// TIA Portal V18 export
FUNCTION_BLOCK "AXIS_CMMT_V2_Motion_Control"   // FB22, LAD
TITLE = Description
{ S7_Optimized_Access := 'TRUE' }
VERSION : 0.1
// This is the motion function block used to control all the axes. Due to some differences in the control part for different types of motion and drives, there are additional conditions in some parts of the code.
// 
// Important things to check if the drive is not moving:
// - homing
// - motion lock from add ons (capping station, no go zones)
// - door sensors
// - operation mode
// - communication with the drives (Online access)
// stored: AutoNumber false, IsIECCheckEnabled false, IsRetainMemResEnabled false, MemoryReserve 100, SetENOAutomatically false, UDAEnableTagReadback false
   VAR_INPUT
      DriverType : String;   // CMMT; CMMS;
      EnableAxis : Bool;
      PrintingModeWebDB : Int;   // Used while executing the movement
      PositionWebDB : DInt;
      VelocityWebDB : Real;
      Stop : Bool;
      EmergencyStop : Bool;
      JogPos : Bool;
      JogNeg : Bool;
      AckError : Bool;
      ConfigEPos : DWord;
      PosMin : DInt;
      PosMax : DInt;
      Jogging : Bool;
      MarginSoft : DInt;
      MarginHard : DInt;
      MotionLock : Bool;   // Axis will not move is this bool is 0
      AXISEnabled : Bool;
      AXISPosOk : Bool;
      AXISReference : Bool;
      AXISAxisWarning : Bool;
      AXISAxisError : Bool;
      AXISLockout : Bool;
      AXISActVelocity : Real;
      AXISActPosition : DInt;
      AXISAxisAckSetpoint : Bool;
      AXISReady4Motion : Bool;
      AXISEposZSW1 : Word;
      AXISStatus : Word;
      JogStartPos : DInt;   // Limit for jogging
      JogEndPos : DInt;   // Limit for jogging
      AxisType : Int;   // Axis Type: 1 - X; 2 - Y; 3 - Z1; 4 - Z2
      YPosition : DInt;
      PositionDelay : Bool;   // Delay to make it easier to confirm that the motion was finished
      NoGoZoneActive : Bool;   // 1 to activate no go zone
      NoGoZoneHomingPermission : Bool;
      NoGoZoneMovePermission : Bool;
      NoGoZoneJogPosPermission : Bool;
      NoGoZoneJogNegPermission : Bool;
      RMPositioningError : DInt := 5;   // Input Relativer Motion Position Error that we accept
      MachineStart : Bool;
   END_VAR
   VAR_OUTPUT
      Status : Word;
      Overrange : Bool;
      Ready : Bool;
      DriveMoving : Bool;
      DriveStop : Bool;
      Standstill : Bool;
      MC : Bool;
      AXISModePos : Int;
      AXISEnableAxis : Bool;
      AXISCancelTraversing : Bool;
      AXISIntermediateStop : Bool;
      AXISJog1 : Bool;
      AXISJog2 : Bool;
      AXISAckError : Bool;
      AXISExecuteMode : Bool;
      AXISPosition : DInt;
      AXISVelocity : Real;
      AXISConfigEpos : DWord;
      AXISRelative : Bool;
      AXISHoming : Bool;
      FinishTask_Delay : Bool;
   END_VAR
   VAR_IN_OUT
      StartTask : Bool;
      Execute : Bool;
      Homing : Bool;
      Printing : Bool;
   END_VAR
   VAR
      ExecutingMemory : Bool;
      HomingMemory : Bool;
      TaskMemory : Bool;
      ModePos : Int := 4;
      PosOk : Bool;
      Reference : Bool;
      PositionInternal : DInt;
      LockoutInternal : Bool;
      RelativeMode : Bool;   // Mode 1
      AbsoluteMode : Bool;   // Mode 2
      TaskFinished : Bool;
      JoggingXPermission : Bool;
      JoggingYPermission : Bool;
      JoggingPOSZ1Z2Permission : Bool;
      JoggingNEGZ1Z2Permission : Bool;
      JoggingPosMax : DInt;
      JoggingPosMin : DInt;
      JoggingPositionCorrection : DInt := 1500;
      ProfinetDisconnected : Bool;
      PositionStepPlus : DInt;
      CMMT : Bool;
      CMMS : Bool;
      RMStepStartPosition : DInt;   // Relative Motion Step Start Position
      RMPredictedPosition : DInt;   // Relative Motion Predicted Position
      RMFinalPosition : DInt;   // Relative Motion Final Position
      RMLastStepPositionError : DInt;   // Relative Motion Last Step Position Error
      RMStartTaskM01 : Bool;   // Relative Motion Start Task M Positive
      RMStartTaksM02 : Bool;   // Relative Motion Start Task M Negative
      RMStepRangePlus : DInt;
      RMStepRangeMinus : DInt;
      RelativeDirectionInRange : Bool;
   END_VAR
   VAR_TEMP
      RelativeModeHomingM : Bool;
      Jog1_pos : Bool;   // Jog positive direction
      Jog2_neg : Bool;   // Jog negative direction
      Memory1 : Bool;
      Memory2 : Bool;
      PosMinSoft : DInt;
      PosMaxSoft : DInt;
      InternalError : Bool;
      InternalWarning : Bool;
      ExecuteBusy : Bool;
      ExecutingInternal : Bool;
      HomingInternal : Bool;
      TaskInternal : Bool;
      Position_Plus : DInt;
      Position_Minus : DInt;
      TestFinished : Bool;
   END_VAR
   VAR CONSTANT
      Position_Error : DInt := 10;
   END_VAR
   VAR_TEMP   // added for the SCL form of the ladder/FBD networks
      _w1 : Bool;
      _w2 : Bool;
      _w3 : Bool;
   END_VAR
BEGIN

REGION Network 1: Checking driver type
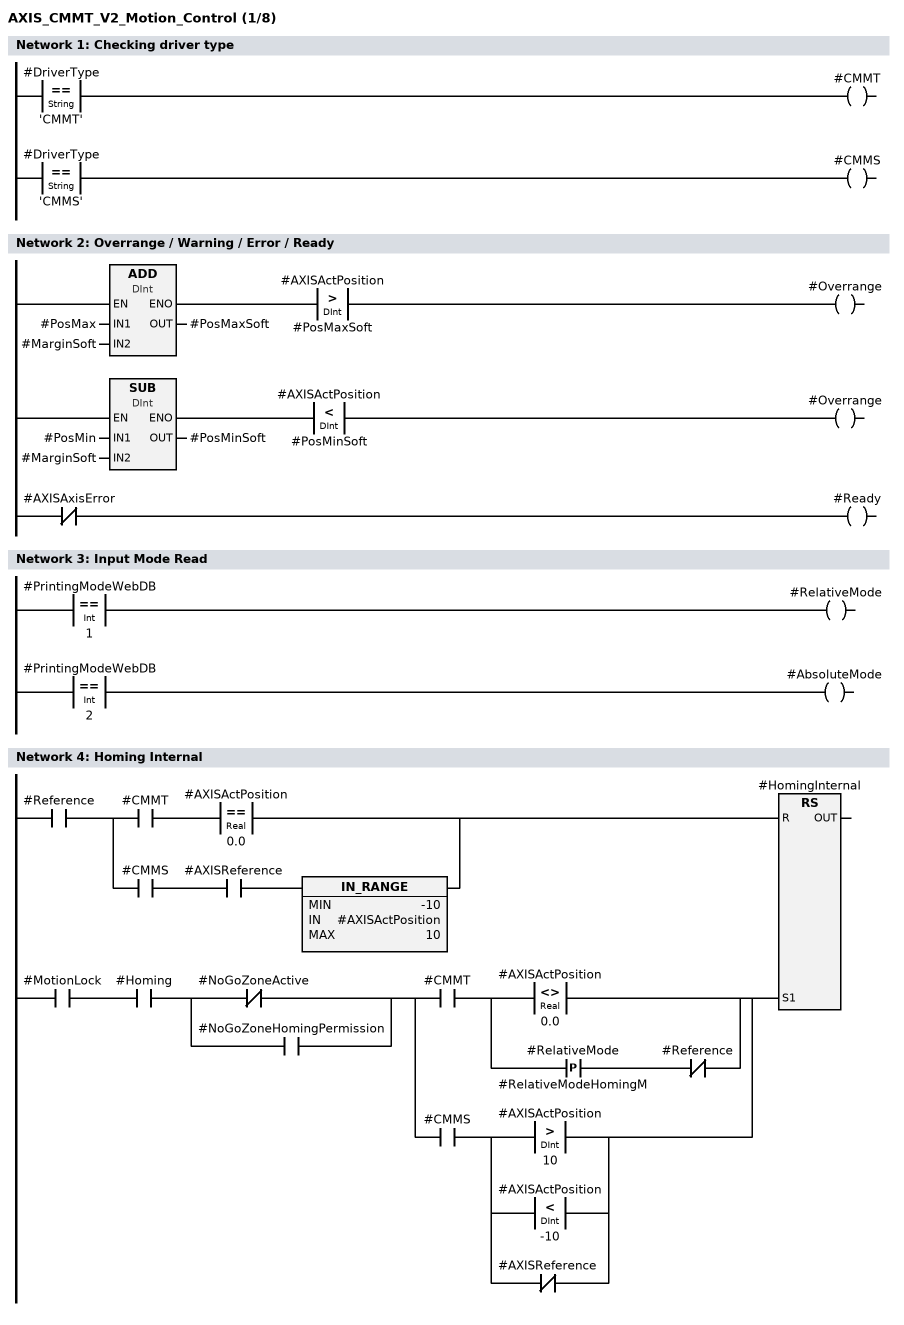
   RUNG wire#powerrail
      { S7_Templates := "SrcType := String" } EQ_Contact(in1 := #DriverType, in2 := 'CMMT')
      Coil( #CMMT )
   END_RUNG
   RUNG wire#powerrail
      { S7_Templates := "SrcType := String" } EQ_Contact(in1 := #DriverType, in2 := 'CMMS')
      Coil( #CMMS )
   END_RUNG
   // the same network as SCL:
   #CMMT := #DriverType = 'CMMT';
   #CMMS := #DriverType = 'CMMS';
END_REGION

REGION Network 2: Overrange / Warning / Error / Ready
   RUNG wire#powerrail
      { S7_Templates := "SrcType := DInt" } Add(in1 := #PosMax, in2 := #MarginSoft, out => #PosMaxSoft)
      { S7_Templates := "SrcType := DInt" } GT_Contact(in1 := #AXISActPosition, in2 := #PosMaxSoft)
      Coil( #Overrange )
   END_RUNG
   RUNG wire#powerrail
      { S7_Templates := "SrcType := DInt" } Sub(in1 := #PosMin, in2 := #MarginSoft, out => #PosMinSoft)
      { S7_Templates := "SrcType := DInt" } LT_Contact(in1 := #AXISActPosition, in2 := #PosMinSoft)
      Coil( #Overrange )
   END_RUNG
   RUNG wire#powerrail
      I_Contact( #AXISAxisError )
      Coil( #Ready )
   END_RUNG
   // the same network as SCL:
   #PosMaxSoft := #PosMax + #MarginSoft;
   #Overrange := #AXISActPosition > #PosMaxSoft;
   #PosMinSoft := #PosMin - #MarginSoft;
   #Overrange := #AXISActPosition < #PosMinSoft;
   #Ready := NOT #AXISAxisError;
END_REGION

REGION Network 3: Input Mode Read
   RUNG wire#powerrail
      { S7_Templates := "SrcType := Int" } EQ_Contact(in1 := #PrintingModeWebDB, in2 := 1)
      Coil( #RelativeMode )
   END_RUNG
   RUNG wire#powerrail
      { S7_Templates := "SrcType := Int" } EQ_Contact(in1 := #PrintingModeWebDB, in2 := 2)
      Coil( #AbsoluteMode )
   END_RUNG
   // the same network as SCL:
   #RelativeMode := #PrintingModeWebDB = 1;
   #AbsoluteMode := #PrintingModeWebDB = 2;
END_REGION

REGION Network 4: Homing Internal
   RUNG wire#powerrail
      Contact( #Reference )
      wire#w1
      Contact( #CMMT )
      { S7_Templates := "SrcType := Real" } EQ_Contact(in1 := #AXISActPosition, in2 := 0.0)
      wire#w2
      S_RS(operand := #HomingInternal, s1 := wire#w7)
   END_RUNG
   RUNG wire#w1
      Contact( #CMMS )
      Contact( #AXISReference )
      { S7_Templates := "SrcType := DInt" } InRange(min := -10, in := #AXISActPosition, max := 10)
   END_RUNG wire#w2
   RUNG wire#powerrail
      Contact( #MotionLock )
      Contact( #Homing )
      wire#w3
      I_Contact( #NoGoZoneActive )
      wire#w4
      Contact( #CMMT )
      wire#w5
      { S7_Templates := "SrcType := Real" } NE_Contact(in1 := #AXISActPosition, in2 := 0.0)
   END_RUNG wire#w7
   RUNG wire#w3
      Contact( #NoGoZoneHomingPermission )
   END_RUNG wire#w4
   RUNG wire#w5
      P_Contact(operand := #RelativeMode, bit := #RelativeModeHomingM)
      I_Contact( #Reference )
   END_RUNG wire#w7
   RUNG wire#w4
      Contact( #CMMS )
      wire#w6
      { S7_Templates := "SrcType := DInt" } GT_Contact(in1 := #AXISActPosition, in2 := 10)
   END_RUNG wire#w7
   RUNG wire#w6
      { S7_Templates := "SrcType := DInt" } LT_Contact(in1 := #AXISActPosition, in2 := -10)
   END_RUNG wire#w7
   RUNG wire#w6
      I_Contact( #AXISReference )
   END_RUNG wire#w7
   // the same network as SCL:
   #_w1 := #MotionLock AND #Homing AND (NOT #NoGoZoneActive OR #NoGoZoneHomingPermission) AND #CMMT AND #RelativeMode AND NOT #RelativeModeHomingM;   // rising edge of #RelativeMode
   #RelativeModeHomingM := #RelativeMode;
   IF #Reference AND ((#CMMT AND (#AXISActPosition = 0.0)) OR (#CMMS AND #AXISReference AND (-10 <= #AXISActPosition) AND (#AXISActPosition <= 10))) THEN
       #HomingInternal := FALSE;   // RS flip-flop
   END_IF;
   IF (#MotionLock AND #Homing AND (NOT #NoGoZoneActive OR #NoGoZoneHomingPermission) AND #CMMT AND (#AXISActPosition <> 0.0)) OR (#_w1 AND NOT #Reference) OR (#MotionLock AND #Homing AND (NOT #NoGoZoneActive OR #NoGoZoneHomingPermission) AND #CMMS AND ((#AXISActPosition > 10) OR (#AXISActPosition < (-10)) OR NOT #AXISReference)) THEN
       #HomingInternal := TRUE;
   END_IF;
END_REGION

REGION Network 5: Status Behavior
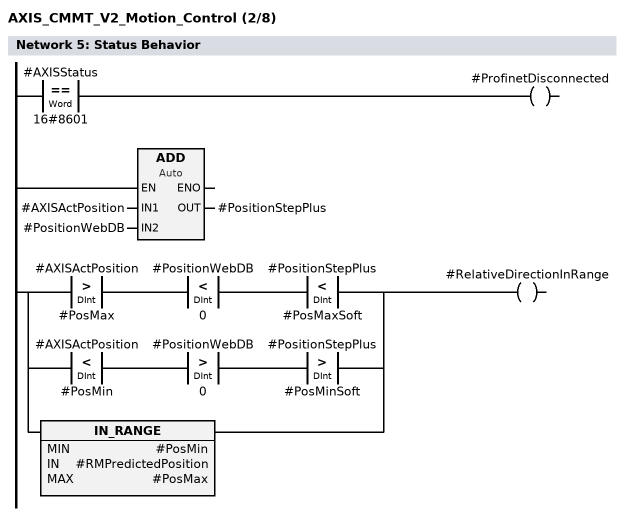
   RUNG wire#powerrail
      { S7_Templates := "SrcType := Word" } EQ_Contact(in1 := #AXISStatus, in2 := 16#8601)
      Coil( #ProfinetDisconnected )
   END_RUNG
   RUNG wire#powerrail
      Add(in1 := #AXISActPosition, in2 := #PositionWebDB, out => #PositionStepPlus)
   END_RUNG
   RUNG wire#powerrail
      { S7_Templates := "SrcType := DInt" } GT_Contact(in1 := #AXISActPosition, in2 := #PosMax)
      { S7_Templates := "SrcType := DInt" } LT_Contact(in1 := #PositionWebDB, in2 := 0)
      { S7_Templates := "SrcType := DInt" } LT_Contact(in1 := #PositionStepPlus, in2 := #PosMaxSoft)
      wire#w1
      Coil( #RelativeDirectionInRange )
   END_RUNG
   RUNG wire#powerrail
      { S7_Templates := "SrcType := DInt" } LT_Contact(in1 := #AXISActPosition, in2 := #PosMin)
      { S7_Templates := "SrcType := DInt" } GT_Contact(in1 := #PositionWebDB, in2 := 0)
      { S7_Templates := "SrcType := DInt" } GT_Contact(in1 := #PositionStepPlus, in2 := #PosMinSoft)
   END_RUNG wire#w1
   RUNG wire#powerrail
      { S7_Templates := "SrcType := DInt" } InRange(min := #PosMin, in := #RMPredictedPosition, max := #PosMax)
   END_RUNG wire#w1
   // the same network as SCL:
   #ProfinetDisconnected := #AXISStatus = 16#8601;
   #PositionStepPlus := #AXISActPosition + #PositionWebDB;
   #RelativeDirectionInRange := ((#AXISActPosition > #PosMax) AND (#PositionWebDB < 0) AND (#PositionStepPlus < #PosMaxSoft)) OR ((#AXISActPosition < #PosMin) AND (#PositionWebDB > 0) AND (#PositionStepPlus > #PosMinSoft)) OR ((#PosMin <= #RMPredictedPosition) AND (#RMPredictedPosition <= #PosMax));
END_REGION

REGION Network 6: Task Internal
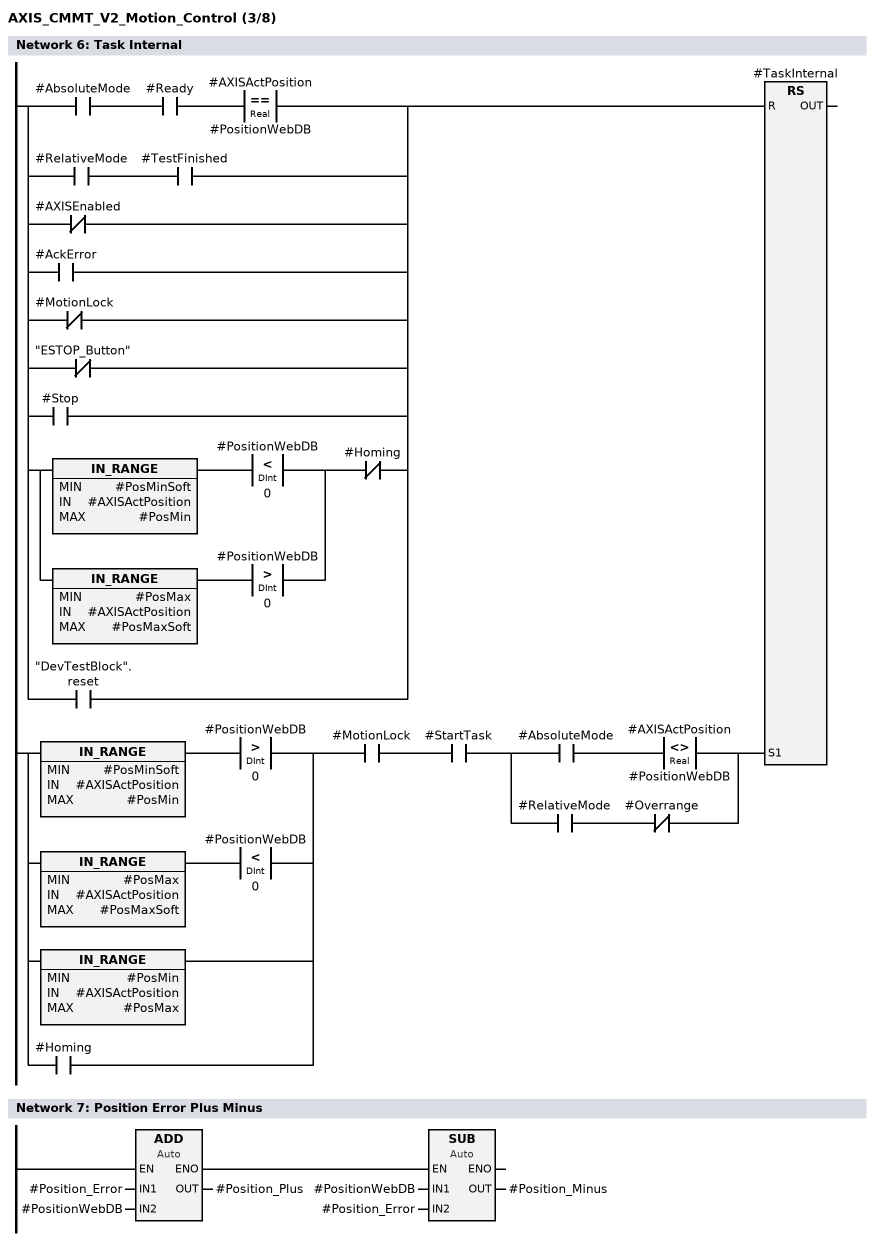
   RUNG wire#powerrail
      Contact( #AbsoluteMode )
      Contact( #Ready )
      { S7_Templates := "SrcType := Real" } EQ_Contact(in1 := #AXISActPosition, in2 := #PositionWebDB)
      wire#w1
      S_RS(operand := #TaskInternal, s1 := wire#w5)
   END_RUNG
   RUNG wire#powerrail
      Contact( #RelativeMode )
      Contact( #TestFinished )
   END_RUNG wire#w1
   RUNG wire#powerrail
      I_Contact( #AXISEnabled )
   END_RUNG wire#w1
   RUNG wire#powerrail
      Contact( #AckError )
   END_RUNG wire#w1
   RUNG wire#powerrail
      I_Contact( #MotionLock )
   END_RUNG wire#w1
   RUNG wire#powerrail
      I_Contact( "ESTOP_Button" )
   END_RUNG wire#w1
   RUNG wire#powerrail
      Contact( #Stop )
   END_RUNG wire#w1
   RUNG wire#powerrail
      { S7_Templates := "SrcType := DInt" } InRange(min := #PosMinSoft, in := #AXISActPosition, max := #PosMin)
      { S7_Templates := "SrcType := DInt" } LT_Contact(in1 := #PositionWebDB, in2 := 0)
      wire#w2
      I_Contact( #Homing )
   END_RUNG wire#w1
   RUNG wire#powerrail
      { S7_Templates := "SrcType := DInt" } InRange(min := #PosMax, in := #AXISActPosition, max := #PosMaxSoft)
      { S7_Templates := "SrcType := DInt" } GT_Contact(in1 := #PositionWebDB, in2 := 0)
   END_RUNG wire#w2
   RUNG wire#powerrail
      Contact( "DevTestBlock".reset )
   END_RUNG wire#w1
   RUNG wire#powerrail
      { S7_Templates := "SrcType := DInt" } InRange(min := #PosMinSoft, in := #AXISActPosition, max := #PosMin)
      { S7_Templates := "SrcType := DInt" } GT_Contact(in1 := #PositionWebDB, in2 := 0)
      wire#w3
      Contact( #MotionLock )
      Contact( #StartTask )
      wire#w4
      Contact( #AbsoluteMode )
      { S7_Templates := "SrcType := Real" } NE_Contact(in1 := #AXISActPosition, in2 := #PositionWebDB)
   END_RUNG wire#w5
   RUNG wire#powerrail
      { S7_Templates := "SrcType := DInt" } InRange(min := #PosMax, in := #AXISActPosition, max := #PosMaxSoft)
      { S7_Templates := "SrcType := DInt" } LT_Contact(in1 := #PositionWebDB, in2 := 0)
   END_RUNG wire#w3
   RUNG wire#powerrail
      { S7_Templates := "SrcType := DInt" } InRange(min := #PosMin, in := #AXISActPosition, max := #PosMax)
   END_RUNG wire#w3
   RUNG wire#powerrail
      Contact( #Homing )
   END_RUNG wire#w3
   RUNG wire#w4
      Contact( #RelativeMode )
      I_Contact( #Overrange )
   END_RUNG wire#w5
   // the same network as SCL:
   IF (#AbsoluteMode AND #Ready AND (#AXISActPosition = #PositionWebDB)) OR (#RelativeMode AND #TestFinished) OR NOT #AXISEnabled OR #AckError OR NOT #MotionLock OR NOT "ESTOP_Button" OR #Stop OR ((((#PosMinSoft <= #AXISActPosition) AND (#AXISActPosition <= #PosMin) AND (#PositionWebDB < 0)) OR ((#PosMax <= #AXISActPosition) AND (#AXISActPosition <= #PosMaxSoft) AND (#PositionWebDB > 0))) AND NOT #Homing) OR "DevTestBlock".reset THEN
       #TaskInternal := FALSE;   // RS flip-flop
   END_IF;
   IF (((#PosMinSoft <= #AXISActPosition) AND (#AXISActPosition <= #PosMin) AND (#PositionWebDB > 0)) OR ((#PosMax <= #AXISActPosition) AND (#AXISActPosition <= #PosMaxSoft) AND (#PositionWebDB < 0)) OR ((#PosMin <= #AXISActPosition) AND (#AXISActPosition <= #PosMax)) OR #Homing) AND #MotionLock AND #StartTask AND ((#AbsoluteMode AND (#AXISActPosition <> #PositionWebDB)) OR (#RelativeMode AND NOT #Overrange)) THEN
       #TaskInternal := TRUE;
   END_IF;
END_REGION

REGION Network 7: Position Error Plus Minus
   RUNG wire#powerrail
      Add(in1 := #Position_Error, in2 := #PositionWebDB, out => #Position_Plus)
      Sub(in1 := #PositionWebDB, in2 := #Position_Error, out => #Position_Minus)
   END_RUNG
   // the same network as SCL:
   #Position_Plus := #Position_Error + #PositionWebDB;
   #Position_Minus := #PositionWebDB - #Position_Error;
END_REGION

REGION Network 8: Execute Internal
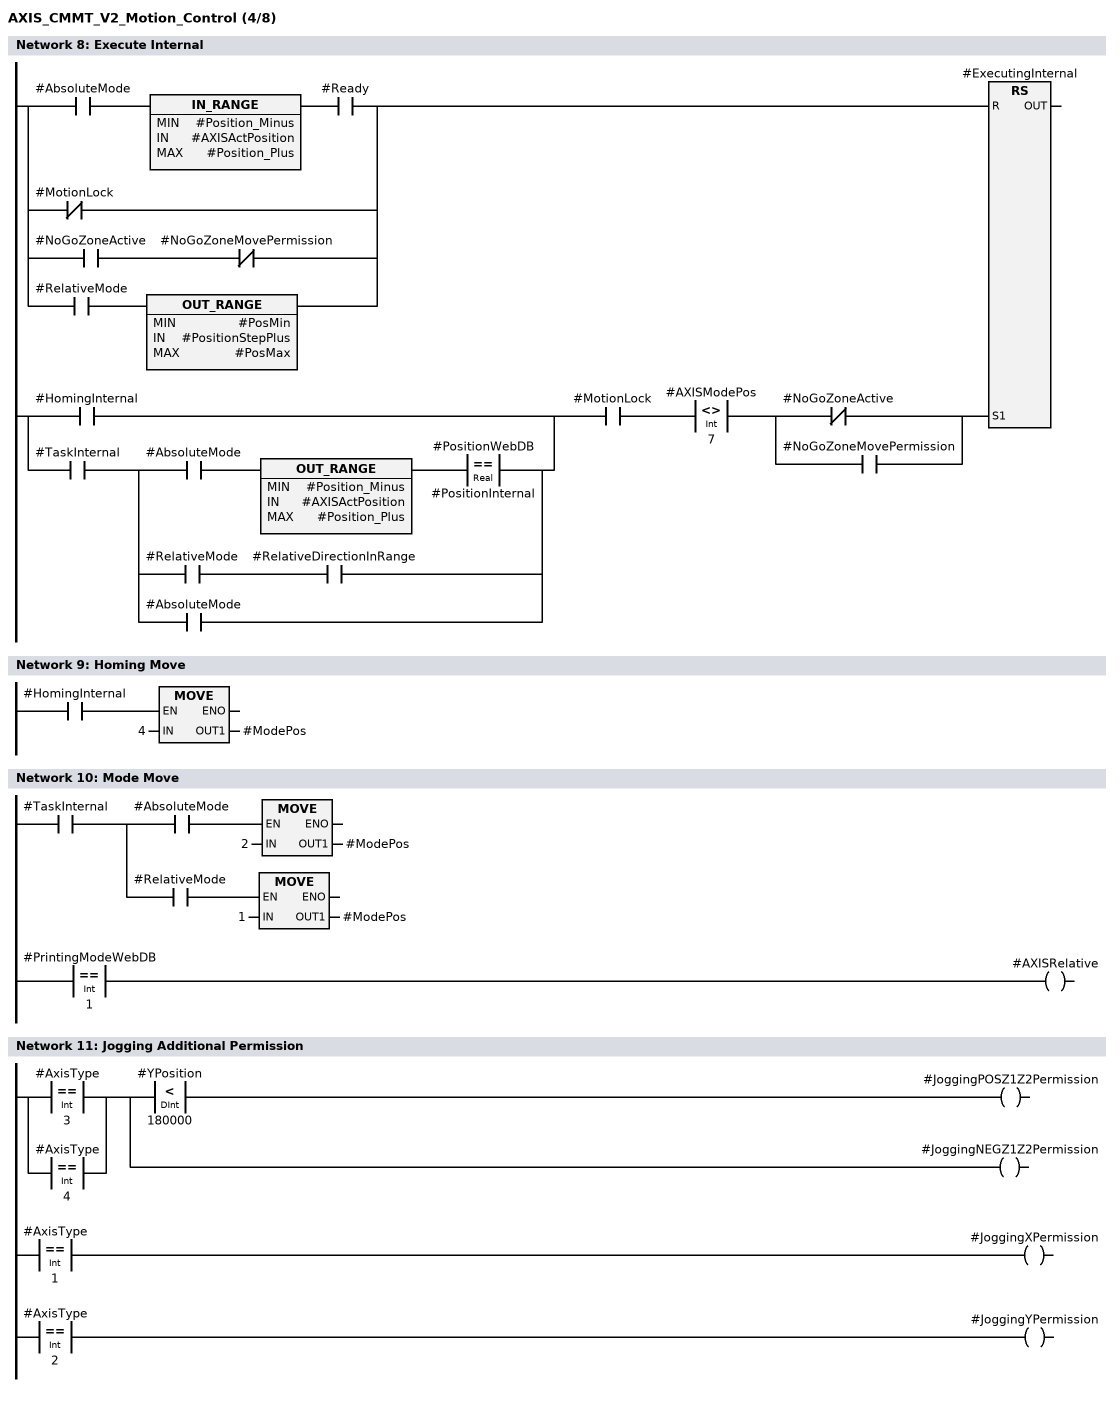
   IF (#AbsoluteMode AND (#Position_Minus <= #AXISActPosition) AND (#AXISActPosition <= #Position_Plus) AND #Ready) OR NOT #MotionLock OR (#NoGoZoneActive AND NOT #NoGoZoneMovePermission) OR (#RelativeMode AND ((#PositionStepPlus < #PosMin) OR (#PositionStepPlus > #PosMax))) THEN
       #ExecutingInternal := FALSE;   // RS flip-flop
   END_IF;
   IF (#HomingInternal OR (#TaskInternal AND ((#AbsoluteMode AND ((#AXISActPosition < #Position_Minus) OR (#AXISActPosition > #Position_Plus)) AND (#PositionWebDB = #PositionInternal)) OR (#RelativeMode AND #RelativeDirectionInRange) OR #AbsoluteMode))) AND #MotionLock AND (#AXISModePos <> 7) AND (NOT #NoGoZoneActive OR #NoGoZoneMovePermission) THEN
       #ExecutingInternal := TRUE;
   END_IF;
END_REGION

REGION Network 9: Homing Move
   RUNG wire#powerrail
      Contact( #HomingInternal )
      Move(in := 4, out1 => #ModePos)
   END_RUNG
   // the same network as SCL:
   IF #HomingInternal THEN #ModePos := 4; END_IF;
END_REGION

REGION Network 10: Mode Move
   RUNG wire#powerrail
      Contact( #TaskInternal )
      wire#w1
      Contact( #AbsoluteMode )
      Move(in := 2, out1 => #ModePos)
   END_RUNG
   RUNG wire#w1
      Contact( #RelativeMode )
      Move(in := 1, out1 => #ModePos)
   END_RUNG
   RUNG wire#powerrail
      { S7_Templates := "SrcType := Int" } EQ_Contact(in1 := #PrintingModeWebDB, in2 := 1)
      Coil( #AXISRelative )
   END_RUNG
   // the same network as SCL:
   IF #TaskInternal AND #AbsoluteMode THEN #ModePos := 2; END_IF;
   IF #TaskInternal AND #RelativeMode THEN #ModePos := 1; END_IF;
   #AXISRelative := #PrintingModeWebDB = 1;
END_REGION

REGION Network 11: Jogging Additional Permission
   RUNG wire#powerrail
      { S7_Templates := "SrcType := Int" } EQ_Contact(in1 := #AxisType, in2 := 3)
      wire#w1
      { S7_Templates := "SrcType := DInt" } LT_Contact(in1 := #YPosition, in2 := 180000)
      Coil( #JoggingPOSZ1Z2Permission )
   END_RUNG
   RUNG wire#powerrail
      { S7_Templates := "SrcType := Int" } EQ_Contact(in1 := #AxisType, in2 := 4)
   END_RUNG wire#w1
   RUNG wire#w1
      Coil( #JoggingNEGZ1Z2Permission )
   END_RUNG
   RUNG wire#powerrail
      { S7_Templates := "SrcType := Int" } EQ_Contact(in1 := #AxisType, in2 := 1)
      Coil( #JoggingXPermission )
   END_RUNG
   RUNG wire#powerrail
      { S7_Templates := "SrcType := Int" } EQ_Contact(in1 := #AxisType, in2 := 2)
      Coil( #JoggingYPermission )
   END_RUNG
   // the same network as SCL:
   #_w1 := (#AxisType = 3) OR (#AxisType = 4);
   #JoggingPOSZ1Z2Permission := #_w1 AND (#YPosition < 180000);
   #JoggingNEGZ1Z2Permission := #_w1;
   #JoggingXPermission := #AxisType = 1;
   #JoggingYPermission := #AxisType = 2;
END_REGION

REGION Network 12: Jogging Limit Change
   // Changed jogging limits to prevent overshooting
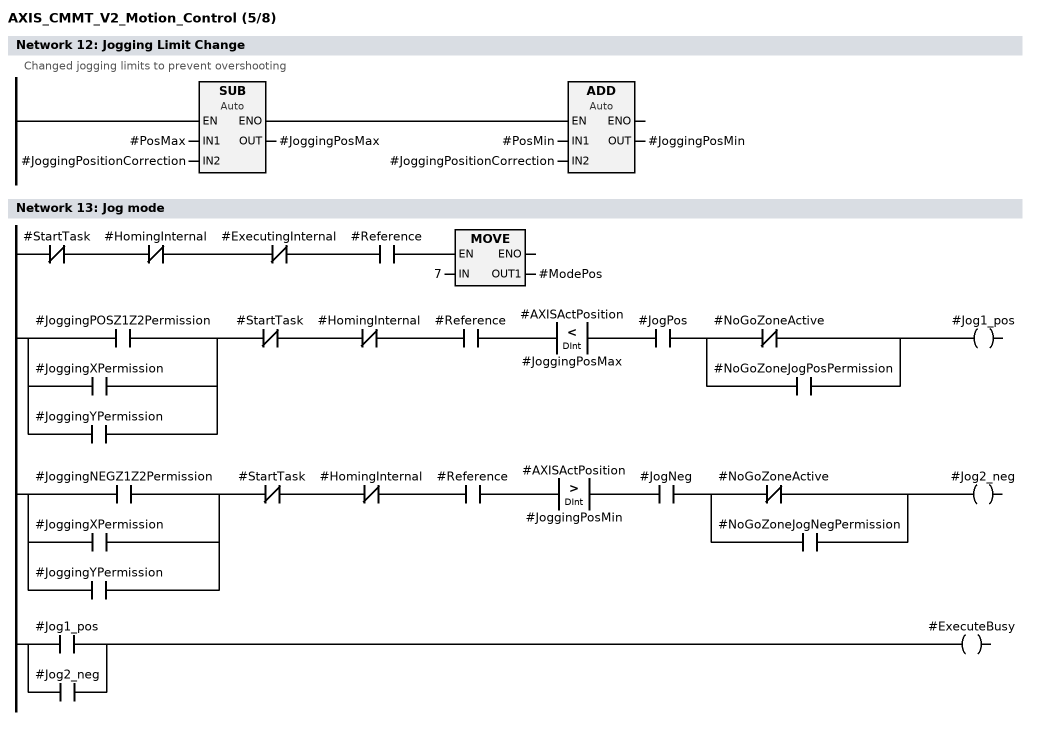
   RUNG wire#powerrail
      Sub(in1 := #PosMax, in2 := #JoggingPositionCorrection, out => #JoggingPosMax)
      Add(in1 := #PosMin, in2 := #JoggingPositionCorrection, out => #JoggingPosMin)
   END_RUNG
   // the same network as SCL:
   #JoggingPosMax := #PosMax - #JoggingPositionCorrection;
   #JoggingPosMin := #PosMin + #JoggingPositionCorrection;
END_REGION

REGION Network 13: Jog mode
   RUNG wire#powerrail
      I_Contact( #StartTask )
      I_Contact( #HomingInternal )
      I_Contact( #ExecutingInternal )
      Contact( #Reference )
      Move(in := 7, out1 => #ModePos)
   END_RUNG
   RUNG wire#powerrail
      Contact( #JoggingPOSZ1Z2Permission )
      wire#w1
      I_Contact( #StartTask )
      I_Contact( #HomingInternal )
      Contact( #Reference )
      { S7_Templates := "SrcType := DInt" } LT_Contact(in1 := #AXISActPosition, in2 := #JoggingPosMax)
      Contact( #JogPos )
      wire#w2
      I_Contact( #NoGoZoneActive )
      wire#w3
      Coil( #Jog1_pos )
   END_RUNG
   RUNG wire#powerrail
      Contact( #JoggingXPermission )
   END_RUNG wire#w1
   RUNG wire#powerrail
      Contact( #JoggingYPermission )
   END_RUNG wire#w1
   RUNG wire#w2
      Contact( #NoGoZoneJogPosPermission )
   END_RUNG wire#w3
   RUNG wire#powerrail
      Contact( #JoggingNEGZ1Z2Permission )
      wire#w4
      I_Contact( #StartTask )
      I_Contact( #HomingInternal )
      Contact( #Reference )
      { S7_Templates := "SrcType := DInt" } GT_Contact(in1 := #AXISActPosition, in2 := #JoggingPosMin)
      Contact( #JogNeg )
      wire#w5
      I_Contact( #NoGoZoneActive )
      wire#w6
      Coil( #Jog2_neg )
   END_RUNG
   RUNG wire#powerrail
      Contact( #JoggingXPermission )
   END_RUNG wire#w4
   RUNG wire#powerrail
      Contact( #JoggingYPermission )
   END_RUNG wire#w4
   RUNG wire#w5
      Contact( #NoGoZoneJogNegPermission )
   END_RUNG wire#w6
   RUNG wire#powerrail
      Contact( #Jog1_pos )
      wire#w7
      Coil( #ExecuteBusy )
   END_RUNG
   RUNG wire#powerrail
      Contact( #Jog2_neg )
   END_RUNG wire#w7
   // the same network as SCL:
   IF NOT #StartTask AND NOT #HomingInternal AND NOT #ExecutingInternal AND #Reference THEN
       #ModePos := 7;
   END_IF;
   #Jog1_pos := (#JoggingPOSZ1Z2Permission OR #JoggingXPermission OR #JoggingYPermission) AND NOT #StartTask AND NOT #HomingInternal AND #Reference AND (#AXISActPosition < #JoggingPosMax) AND #JogPos AND (NOT #NoGoZoneActive OR #NoGoZoneJogPosPermission);
   #Jog2_neg := (#JoggingNEGZ1Z2Permission OR #JoggingXPermission OR #JoggingYPermission) AND NOT #StartTask AND NOT #HomingInternal AND #Reference AND (#AXISActPosition > #JoggingPosMin) AND #JogNeg AND (NOT #NoGoZoneActive OR #NoGoZoneJogNegPermission);
   #ExecuteBusy := #Jog1_pos OR #Jog2_neg;
END_REGION

REGION Network 14: Motion Block Control
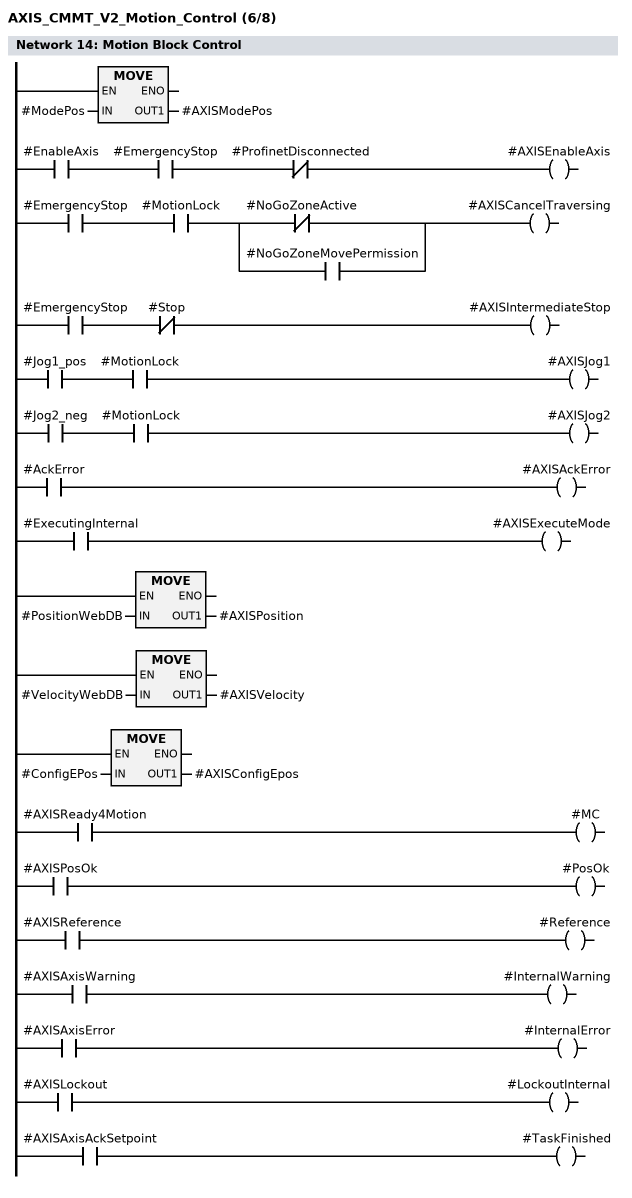
   RUNG wire#powerrail
      Move(in := #ModePos, out1 => #AXISModePos)
   END_RUNG
   RUNG wire#powerrail
      Contact( #EnableAxis )
      Contact( #EmergencyStop )
      I_Contact( #ProfinetDisconnected )
      Coil( #AXISEnableAxis )
   END_RUNG
   RUNG wire#powerrail
      Contact( #EmergencyStop )
      Contact( #MotionLock )
      wire#w1
      I_Contact( #NoGoZoneActive )
      wire#w2
      Coil( #AXISCancelTraversing )
   END_RUNG
   RUNG wire#w1
      Contact( #NoGoZoneMovePermission )
   END_RUNG wire#w2
   RUNG wire#powerrail
      Contact( #EmergencyStop )
      I_Contact( #Stop )
      Coil( #AXISIntermediateStop )
   END_RUNG
   RUNG wire#powerrail
      Contact( #Jog1_pos )
      Contact( #MotionLock )
      Coil( #AXISJog1 )
   END_RUNG
   RUNG wire#powerrail
      Contact( #Jog2_neg )
      Contact( #MotionLock )
      Coil( #AXISJog2 )
   END_RUNG
   RUNG wire#powerrail
      Contact( #AckError )
      Coil( #AXISAckError )
   END_RUNG
   RUNG wire#powerrail
      Contact( #ExecutingInternal )
      Coil( #AXISExecuteMode )
   END_RUNG
   RUNG wire#powerrail
      Move(in := #PositionWebDB, out1 => #AXISPosition)
   END_RUNG
   RUNG wire#powerrail
      Move(in := #VelocityWebDB, out1 => #AXISVelocity)
   END_RUNG
   RUNG wire#powerrail
      Move(in := #ConfigEPos, out1 => #AXISConfigEpos)
   END_RUNG
   RUNG wire#powerrail
      Contact( #AXISReady4Motion )
      Coil( #MC )
   END_RUNG
   RUNG wire#powerrail
      Contact( #AXISPosOk )
      Coil( #PosOk )
   END_RUNG
   RUNG wire#powerrail
      Contact( #AXISReference )
      Coil( #Reference )
   END_RUNG
   RUNG wire#powerrail
      Contact( #AXISAxisWarning )
      Coil( #InternalWarning )
   END_RUNG
   RUNG wire#powerrail
      Contact( #AXISAxisError )
      Coil( #InternalError )
   END_RUNG
   RUNG wire#powerrail
      Contact( #AXISLockout )
      Coil( #LockoutInternal )
   END_RUNG
   RUNG wire#powerrail
      Contact( #AXISAxisAckSetpoint )
      Coil( #TaskFinished )
   END_RUNG
   // the same network as SCL:
   #AXISModePos := #ModePos;
   #AXISEnableAxis := #EnableAxis AND #EmergencyStop AND NOT #ProfinetDisconnected;
   #AXISCancelTraversing := #EmergencyStop AND #MotionLock AND (NOT #NoGoZoneActive OR #NoGoZoneMovePermission);
   #AXISIntermediateStop := #EmergencyStop AND NOT #Stop;
   #AXISJog1 := #Jog1_pos AND #MotionLock;
   #AXISJog2 := #Jog2_neg AND #MotionLock;
   #AXISAckError := #AckError;
   #AXISExecuteMode := #ExecutingInternal;
   #AXISPosition := #PositionWebDB;
   #AXISVelocity := #VelocityWebDB;
   #AXISConfigEpos := #ConfigEPos;
   #MC := #AXISReady4Motion;
   #PosOk := #AXISPosOk;
   #Reference := #AXISReference;
   #InternalWarning := #AXISAxisWarning;
   #InternalError := #AXISAxisError;
   #LockoutInternal := #AXISLockout;
   #TaskFinished := #AXISAxisAckSetpoint;
END_REGION

REGION Network 15: Mem
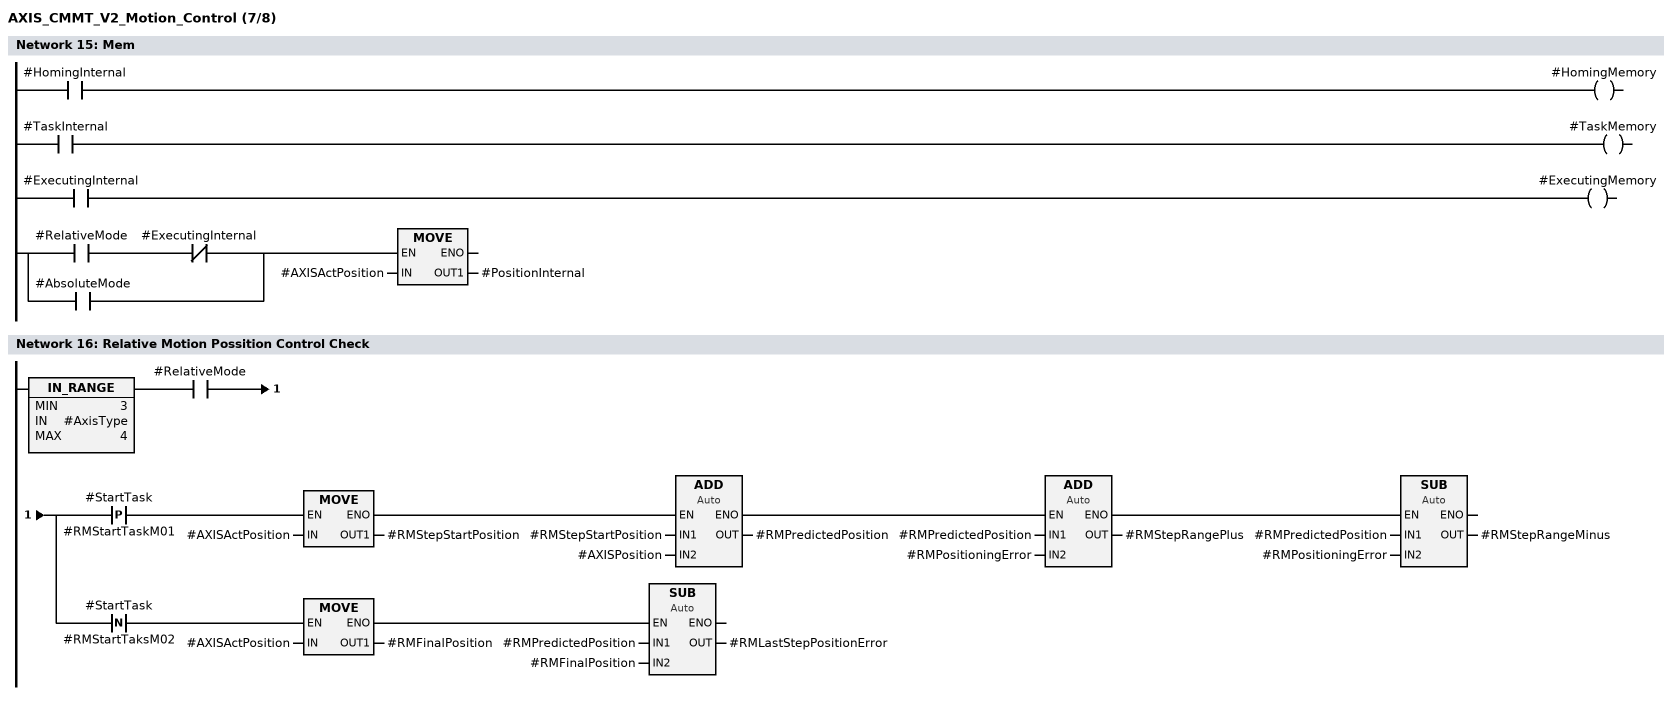
   RUNG wire#powerrail
      Contact( #HomingInternal )
      Coil( #HomingMemory )
   END_RUNG
   RUNG wire#powerrail
      Contact( #TaskInternal )
      Coil( #TaskMemory )
   END_RUNG
   RUNG wire#powerrail
      Contact( #ExecutingInternal )
      Coil( #ExecutingMemory )
   END_RUNG
   RUNG wire#powerrail
      Contact( #RelativeMode )
      I_Contact( #ExecutingInternal )
      wire#w1
      Move(in := #AXISActPosition, out1 => #PositionInternal)
   END_RUNG
   RUNG wire#powerrail
      Contact( #AbsoluteMode )
   END_RUNG wire#w1
   // the same network as SCL:
   #HomingMemory := #HomingInternal;
   #TaskMemory := #TaskInternal;
   #ExecutingMemory := #ExecutingInternal;
   IF (#RelativeMode AND NOT #ExecutingInternal) OR #AbsoluteMode THEN
       #PositionInternal := #AXISActPosition;
   END_IF;
END_REGION

REGION Network 16: Relative Motion Possition Control Check
   RUNG wire#powerrail
      { S7_Templates := "SrcType := Int" } InRange(min := 3, in := #AxisType, max := 4)
      Contact( #RelativeMode )
      wire#w1
      P_Contact(operand := #StartTask, bit := #RMStartTaskM01)
      Move(in := #AXISActPosition, out1 => #RMStepStartPosition)
      Add(in1 := #RMStepStartPosition, in2 := #AXISPosition, out => #RMPredictedPosition)
      Add(in1 := #RMPredictedPosition, in2 := #RMPositioningError, out => #RMStepRangePlus)
      Sub(in1 := #RMPredictedPosition, in2 := #RMPositioningError, out => #RMStepRangeMinus)
   END_RUNG
   RUNG wire#w1
      N_Contact(operand := #StartTask, bit := #RMStartTaksM02)
      Move(in := #AXISActPosition, out1 => #RMFinalPosition)
      Sub(in1 := #RMPredictedPosition, in2 := #RMFinalPosition, out => #RMLastStepPositionError)
   END_RUNG
   // the same network as SCL:
   #_w1 := (3 <= #AxisType) AND (#AxisType <= 4) AND #RelativeMode;
   #_w2 := #_w1 AND #StartTask AND NOT #RMStartTaskM01;   // rising edge of #StartTask
   #RMStartTaskM01 := #StartTask;
   IF #_w2 THEN
       #RMStepStartPosition := #AXISActPosition;
       #RMPredictedPosition := #RMStepStartPosition + #AXISPosition;
       #RMStepRangePlus := #RMPredictedPosition + #RMPositioningError;
       #RMStepRangeMinus := #RMPredictedPosition - #RMPositioningError;
   END_IF;
   #_w3 := #_w1 AND NOT #StartTask AND #RMStartTaksM02;   // falling edge of #StartTask
   #RMStartTaksM02 := #StartTask;
   IF #_w3 THEN
       #RMFinalPosition := #AXISActPosition;
       #RMLastStepPositionError := #RMPredictedPosition - #RMFinalPosition;
   END_IF;
END_REGION

REGION Network 17: Status Move
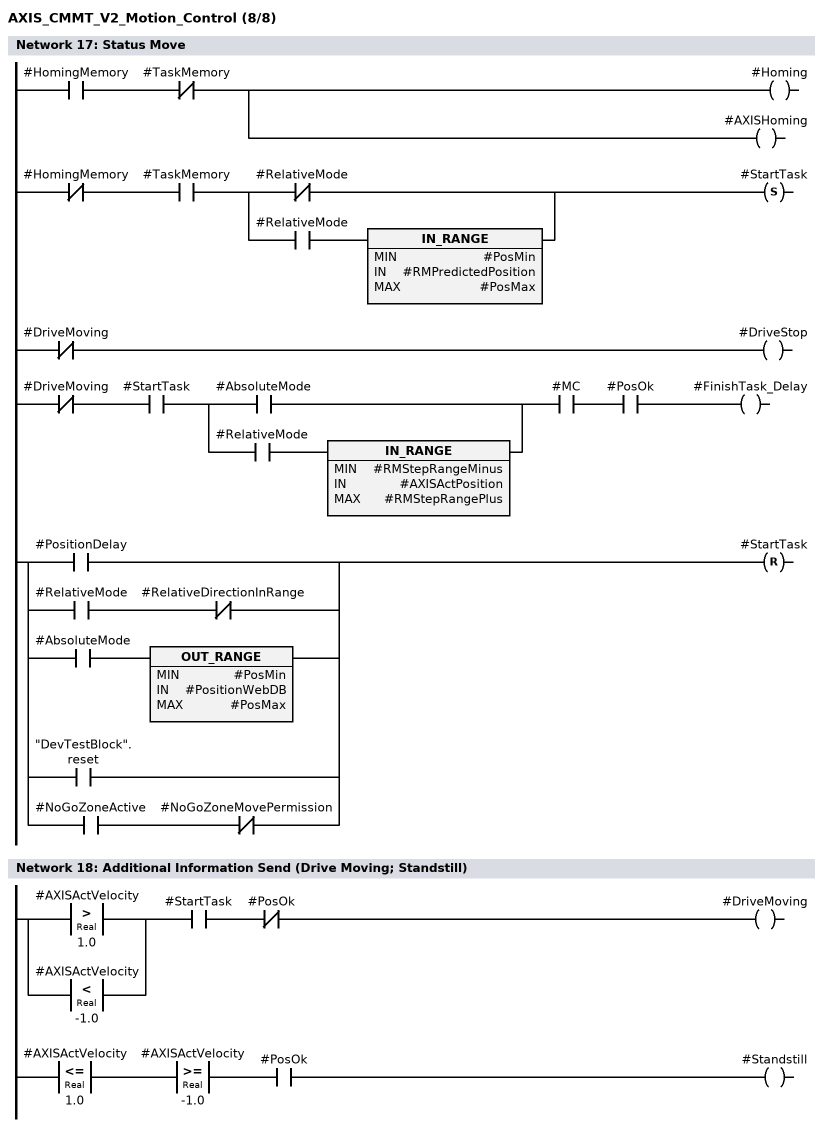
   #Homing := #HomingMemory AND NOT #TaskMemory;
   #AXISHoming := #Homing;
   IF NOT #HomingMemory AND #TaskMemory AND (NOT #RelativeMode OR (#RelativeMode AND (#PosMin <= #RMPredictedPosition) AND (#RMPredictedPosition <= #PosMax))) THEN
       #StartTask := TRUE;
   END_IF;
   #DriveStop := NOT #DriveMoving;
   #FinishTask_Delay := NOT #DriveMoving AND #StartTask AND (#AbsoluteMode OR (#RelativeMode AND (#RMStepRangeMinus <= #AXISActPosition) AND (#AXISActPosition <= #RMStepRangePlus))) AND #MC AND #PosOk;
   IF #PositionDelay OR (#RelativeMode AND NOT #RelativeDirectionInRange) OR (#AbsoluteMode AND ((#PositionWebDB < #PosMin) OR (#PositionWebDB > #PosMax))) OR "DevTestBlock".reset OR (#NoGoZoneActive AND NOT #NoGoZoneMovePermission) THEN
       #StartTask := FALSE;
   END_IF;
END_REGION

REGION Network 18: Additional Information Send (Drive Moving; Standstill)
   RUNG wire#powerrail
      { S7_Templates := "SrcType := Real" } GT_Contact(in1 := #AXISActVelocity, in2 := 1.0)
      wire#w1
      Contact( #StartTask )
      I_Contact( #PosOk )
      Coil( #DriveMoving )
   END_RUNG
   RUNG wire#powerrail
      { S7_Templates := "SrcType := Real" } LT_Contact(in1 := #AXISActVelocity, in2 := -1.0)
   END_RUNG wire#w1
   RUNG wire#powerrail
      { S7_Templates := "SrcType := Real" } LE_Contact(in1 := #AXISActVelocity, in2 := 1.0)
      { S7_Templates := "SrcType := Real" } GE_Contact(in1 := #AXISActVelocity, in2 := -1.0)
      Contact( #PosOk )
      Coil( #Standstill )
   END_RUNG
   // the same network as SCL:
   #DriveMoving := ((#AXISActVelocity > 1.0) OR (#AXISActVelocity < (-1.0))) AND #StartTask AND NOT #PosOk;
   #Standstill := (#AXISActVelocity <= 1.0) AND (#AXISActVelocity >= (-1.0)) AND #PosOk;
END_REGION
END_FUNCTION_BLOCK
